{attribute addProperty BoxType "EK1100-0000-0018"}
{attribute addProperty Id "Beckhoff_EL34xxEK1122Beckhoff_EL34xxEK1122_54E02F3C162A_0001_EL3403_0000_0017EL3403_CEBF0ECD61677A_0002_EL3403_0000_0018EL3403_0856E9FD61677A_0003_EL3403_0000_0019EL3403_0856E9FD61677A_0004_EL3403_0000_0020EL3403_0856E9FD61677A_0005_EL3403_0000_0021EL3403_0856E9FD61677A_0006_EL3403_0000_0022EL3403_26274D9958473A_0007_EL3403_0000_0023EL3403_26274D9958473A_0008_EL3403_0010_0017EL3403_CEBF0ECD61677A_0009_EL3403_0010_0018EL3403_0856E9FD61677A_0010_EL3403_0010_0019EL3403_0856E9FD61677A_0011_EL3403_0010_0020EL3403_0856E9FD61677A_0012_EL3403_0010_0021EL3403_0856E9FD61677A_0013_EL3403_0010_0022EL3403_26274D9958473A_0014_EL3403_0010_0023EL3403_26274D9958473A_0015_EL3403_0010_0024EL3403_26274D9958473A_0016_EL3403_0026_0017EL3403_CEBF0ECD61677A_0017_EL3403_0026_0018EL3403_0856E9FD61677A_0018_EL3403_0026_0019EL3403_0856E9FD61677A_0019_EL3403_0026_0020EL3403_0856E9FD61677A_0020_EL3403_0026_0021EL3403_0856E9FD61677A_0021_EL3403_0026_0022EL3403_26274D9958473A_0022_EL3403_0026_0023EL3403_26274D9958473A_0023_EL3403_0026_0024EL3403_26274D9958473A_0024_EL3403_0100_0017EL3403_CEBF0ECD61677A_0025_EL3403_0100_0018EL3403_0856E9FD61677A_0026_EL3403_0100_0019EL3403_0856E9FD61677A_0027_EL3403_0100_0020EL3403_0856E9FD61677A_0028_EL3403_0100_0021EL3403_0856E9FD61677A_0029_EL3403_0100_0022EL3403_26274D9958473A_0030_EL3403_0100_0023EL3403_26274D9958473A_0031_EL3403_0100_0024EL3403_26274D9958473A_0032_EL3403_0111_0017EL3403_CEBF0ECD61677A_0033_EL3403_0111_0018EL3403_0856E9FD61677A_0034_EL3403_0111_0019EL3403_0856E9FD61677A_0035_EL3403_0111_0020EL3403_0856E9FD61677A_0036_EL3403_0111_0021EL3403_0856E9FD61677A_0037_EL3403_0111_0022EL3403_26274D9958473A_0038_EL3403_0111_0023EL3403_26274D9958473A_0039_EL3403_0111_0024EL3403_26274D9958473A_0040_EL3403_0126_0017EL3403_CEBF0ECD61677A_0041_EL3403_0126_0018EL3403_0856E9FD61677A_0042_EL3403_0126_0019EL3403_0856E9FD61677A_0043_EL3403_0126_0020EL3403_0856E9FD61677A_0044_EL3403_0126_0021EL3403_0856E9FD61677A_0045_EL3403_0126_0022EL3403_26274D9958473A_0046_EL3403_0126_0023EL3403_26274D9958473A_0047_EL3403_0126_0024EL3403_26274D9958473A_0048_EL3403_0333_0023EL3403_26274D9958473A_0049_EL3403_0333_0024EL3403_26274D9958473A_0050_EL3413_0000_0016EL3413_446C23E765682A_0051_EL3413_0000_0017EL3413_446C23E765682A_0052_EL3413_0000_0018EL3413_446C23E765682A_0053_EL3413_0000_0019EL3413_7AF41FD265682A_0054_EL3413_0000_0020EL3413_7AF41FD265682A_0055_EL3413_0001_0016EL3413_7AF41FD265682A_0056_EL3413_0001_0017EL3413_7AF41FD265682A_0057_EL3413_0120_0017EL3413_446C23E765682A_0058_EL3413_0001_0018EL3413_7AF41FD265682A_0059_EL3413_0120_0018EL3413_7AF41FD265682A_0060_EL3413_0120_0019EL3413_7AF41FD265682A_0061_EL3423_0000_0016EL3423_A72AC4D21520190A_0062_EL3423_0000_0017EL3423_51F4B0921520190A_0063_EL3423_0000_0018EL3423_51F4B0921520190A_0064_EL3423_0000_0019EL3423_51F4B0921520190A_0065_EL3423_0000_0020EL3423_5F1A409A944118A_0066_EL3423_0000_0021EL3423_5F1A409A944118A_0067_EL3433_0000_0016EL3433_7AF41FD265682A_0068_EL3433_0000_0017EL3433_7AF41FD265682A_0069_EL3433_0000_0018EL3433_7AF41FD265682A_0070_EL3443_0000_0016EL3443_FBA7AEAF1664208A_0071_EL3443_0000_0017EL3443_A40FED4E1664208A_0072_EL3443_0000_0018EL3443_A40FED4E1664208A_0073_EL3443_0000_0019EL3443_A40FED4E1664208A_0074_EL3443_0000_0020EL3443_FBA7AEAF1664208A_0075_EL3443_0000_0021EL3443_FBA7AEAF1664208A_0076_EL3443_0010_0016EL3443_FBA7AEAF1664208A_0077_EL3443_0010_0017EL3443_A40FED4E1664208A_0078_EL3443_0010_0018EL3443_A40FED4E1664208A_0079_EL3443_0010_0019EL3443_A40FED4E1664208A_0080_EL3443_0010_0020EL3443_FBA7AEAF1664208A_0081_EL3443_0010_0021EL3443_FBA7AEAF1664208A_0082_EL3443_0011_0018EL3443_A40FED4E1664208A_0083_EL3443_0011_0019EL3443_A40FED4E1664208A_0084_EL3443_0011_0020EL3443_FBA7AEAF1664208A_0085_EL3443_0011_0021EL3443_FBA7AEAF1664208A_0086_EL3443_0013_0018EL3443_A40FED4E1664208A_0087_EL3443_0013_0019EL3443_A40FED4E1664208A_0088_EL3443_0013_0020EL3443_FBA7AEAF1664208A_0089_EL3443_0013_0021EL3443_FBA7AEAF1664208A_0090_EL3446_0000_0016EL3446_CF28416359274A_0091_EL3446_0000_0017EL3446_CF28416359274A_0092_EL3453_0000_0017EL3453_04D436851216152A_0093_EL3453_0000_0018EL3453_0BDF0D211208151A_0094_EL3453_0000_0019EL3453_0BDF0D211208151A_0095_EL3453_0000_0020EL3453_04D436851216152A_0096_EL3453_0000_0021EL3453_04D436851216152A_0097_EL3453_0100_0021EL3453_04D436851216152A_0098_EL3483_0000_0016EL3483_4775AA5232841A_0099_EL3483_0000_0017EL3483_4775AA5232841A_0100_EL3483_0000_0018EL3483_4775AA5232841A_0101_EL3483_0000_0019EL3483_4775AA5232841A_0102_EL3483_0000_0020EL3483_4775AA5232841A_0103_EL3483_0000_0021EL3483_4775AA5232841A_0104_EL3483_0060_0018EL3483_52D9841A52065A_0105_EL3483_0060_0019EL3483_52D9841A52065A_0106_EL3483_0060_0020EL3483_FF2A77B352065A_0107_EL3483_0060_0021EL3483_FF2A77B352065"}
{attribute addProperty CRC "1912410272"}
{attribute addProperty SizeInBites "92536"}
{attribute addProperty SizeInBytes "11567"}
TYPE Beckhoff_EL34xx_71FD10A0 EXTENDS EK1100_179A0949 :
STRUCT
	{attribute addProperty Name "Beckhoff_EL34xxEK1122"}
	Beckhoff_EL34xxEK1122 : Beckhoff_EL34xxEK1122_54E02F3C;
	{attribute addProperty Name "A_0001_EL3403_0000_0017"}
	A_0001_EL3403_0000_0017 : EL3403_CEBF0ECD;
	{attribute addProperty Name "A_0002_EL3403_0000_0018"}
	A_0002_EL3403_0000_0018 : EL3403_0856E9FD;
	{attribute addProperty Name "A_0003_EL3403_0000_0019"}
	A_0003_EL3403_0000_0019 : EL3403_0856E9FD;
	{attribute addProperty Name "A_0004_EL3403_0000_0020"}
	A_0004_EL3403_0000_0020 : EL3403_0856E9FD;
	{attribute addProperty Name "A_0005_EL3403_0000_0021"}
	A_0005_EL3403_0000_0021 : EL3403_0856E9FD;
	{attribute addProperty Name "A_0006_EL3403_0000_0022"}
	A_0006_EL3403_0000_0022 : EL3403_26274D99;
	{attribute addProperty Name "A_0007_EL3403_0000_0023"}
	A_0007_EL3403_0000_0023 : EL3403_26274D99;
	{attribute addProperty Name "A_0008_EL3403_0010_0017"}
	A_0008_EL3403_0010_0017 : EL3403_CEBF0ECD;
	{attribute addProperty Name "A_0009_EL3403_0010_0018"}
	A_0009_EL3403_0010_0018 : EL3403_0856E9FD;
	{attribute addProperty Name "A_0010_EL3403_0010_0019"}
	A_0010_EL3403_0010_0019 : EL3403_0856E9FD;
	{attribute addProperty Name "A_0011_EL3403_0010_0020"}
	A_0011_EL3403_0010_0020 : EL3403_0856E9FD;
	{attribute addProperty Name "A_0012_EL3403_0010_0021"}
	A_0012_EL3403_0010_0021 : EL3403_0856E9FD;
	{attribute addProperty Name "A_0013_EL3403_0010_0022"}
	A_0013_EL3403_0010_0022 : EL3403_26274D99;
	{attribute addProperty Name "A_0014_EL3403_0010_0023"}
	A_0014_EL3403_0010_0023 : EL3403_26274D99;
	{attribute addProperty Name "A_0015_EL3403_0010_0024"}
	A_0015_EL3403_0010_0024 : EL3403_26274D99;
	{attribute addProperty Name "A_0016_EL3403_0026_0017"}
	A_0016_EL3403_0026_0017 : EL3403_CEBF0ECD;
	{attribute addProperty Name "A_0017_EL3403_0026_0018"}
	A_0017_EL3403_0026_0018 : EL3403_0856E9FD;
	{attribute addProperty Name "A_0018_EL3403_0026_0019"}
	A_0018_EL3403_0026_0019 : EL3403_0856E9FD;
	{attribute addProperty Name "A_0019_EL3403_0026_0020"}
	A_0019_EL3403_0026_0020 : EL3403_0856E9FD;
	{attribute addProperty Name "A_0020_EL3403_0026_0021"}
	A_0020_EL3403_0026_0021 : EL3403_0856E9FD;
	{attribute addProperty Name "A_0021_EL3403_0026_0022"}
	A_0021_EL3403_0026_0022 : EL3403_26274D99;
	{attribute addProperty Name "A_0022_EL3403_0026_0023"}
	A_0022_EL3403_0026_0023 : EL3403_26274D99;
	{attribute addProperty Name "A_0023_EL3403_0026_0024"}
	A_0023_EL3403_0026_0024 : EL3403_26274D99;
	{attribute addProperty Name "A_0024_EL3403_0100_0017"}
	A_0024_EL3403_0100_0017 : EL3403_CEBF0ECD;
	{attribute addProperty Name "A_0025_EL3403_0100_0018"}
	A_0025_EL3403_0100_0018 : EL3403_0856E9FD;
	{attribute addProperty Name "A_0026_EL3403_0100_0019"}
	A_0026_EL3403_0100_0019 : EL3403_0856E9FD;
	{attribute addProperty Name "A_0027_EL3403_0100_0020"}
	A_0027_EL3403_0100_0020 : EL3403_0856E9FD;
	{attribute addProperty Name "A_0028_EL3403_0100_0021"}
	A_0028_EL3403_0100_0021 : EL3403_0856E9FD;
	{attribute addProperty Name "A_0029_EL3403_0100_0022"}
	A_0029_EL3403_0100_0022 : EL3403_26274D99;
	{attribute addProperty Name "A_0030_EL3403_0100_0023"}
	A_0030_EL3403_0100_0023 : EL3403_26274D99;
	{attribute addProperty Name "A_0031_EL3403_0100_0024"}
	A_0031_EL3403_0100_0024 : EL3403_26274D99;
	{attribute addProperty Name "A_0032_EL3403_0111_0017"}
	A_0032_EL3403_0111_0017 : EL3403_CEBF0ECD;
	{attribute addProperty Name "A_0033_EL3403_0111_0018"}
	A_0033_EL3403_0111_0018 : EL3403_0856E9FD;
	{attribute addProperty Name "A_0034_EL3403_0111_0019"}
	A_0034_EL3403_0111_0019 : EL3403_0856E9FD;
	{attribute addProperty Name "A_0035_EL3403_0111_0020"}
	A_0035_EL3403_0111_0020 : EL3403_0856E9FD;
	{attribute addProperty Name "A_0036_EL3403_0111_0021"}
	A_0036_EL3403_0111_0021 : EL3403_0856E9FD;
	{attribute addProperty Name "A_0037_EL3403_0111_0022"}
	A_0037_EL3403_0111_0022 : EL3403_26274D99;
	{attribute addProperty Name "A_0038_EL3403_0111_0023"}
	A_0038_EL3403_0111_0023 : EL3403_26274D99;
	{attribute addProperty Name "A_0039_EL3403_0111_0024"}
	A_0039_EL3403_0111_0024 : EL3403_26274D99;
	{attribute addProperty Name "A_0040_EL3403_0126_0017"}
	A_0040_EL3403_0126_0017 : EL3403_CEBF0ECD;
	{attribute addProperty Name "A_0041_EL3403_0126_0018"}
	A_0041_EL3403_0126_0018 : EL3403_0856E9FD;
	{attribute addProperty Name "A_0042_EL3403_0126_0019"}
	A_0042_EL3403_0126_0019 : EL3403_0856E9FD;
	{attribute addProperty Name "A_0043_EL3403_0126_0020"}
	A_0043_EL3403_0126_0020 : EL3403_0856E9FD;
	{attribute addProperty Name "A_0044_EL3403_0126_0021"}
	A_0044_EL3403_0126_0021 : EL3403_0856E9FD;
	{attribute addProperty Name "A_0045_EL3403_0126_0022"}
	A_0045_EL3403_0126_0022 : EL3403_26274D99;
	{attribute addProperty Name "A_0046_EL3403_0126_0023"}
	A_0046_EL3403_0126_0023 : EL3403_26274D99;
	{attribute addProperty Name "A_0047_EL3403_0126_0024"}
	A_0047_EL3403_0126_0024 : EL3403_26274D99;
	{attribute addProperty Name "A_0048_EL3403_0333_0023"}
	A_0048_EL3403_0333_0023 : EL3403_26274D99;
	{attribute addProperty Name "A_0049_EL3403_0333_0024"}
	A_0049_EL3403_0333_0024 : EL3403_26274D99;
	{attribute addProperty Name "A_0050_EL3413_0000_0016"}
	A_0050_EL3413_0000_0016 : EL3413_446C23E7;
	{attribute addProperty Name "A_0051_EL3413_0000_0017"}
	A_0051_EL3413_0000_0017 : EL3413_446C23E7;
	{attribute addProperty Name "A_0052_EL3413_0000_0018"}
	A_0052_EL3413_0000_0018 : EL3413_446C23E7;
	{attribute addProperty Name "A_0053_EL3413_0000_0019"}
	A_0053_EL3413_0000_0019 : EL3413_7AF41FD2;
	{attribute addProperty Name "A_0054_EL3413_0000_0020"}
	A_0054_EL3413_0000_0020 : EL3413_7AF41FD2;
	{attribute addProperty Name "A_0055_EL3413_0001_0016"}
	A_0055_EL3413_0001_0016 : EL3413_7AF41FD2;
	{attribute addProperty Name "A_0056_EL3413_0001_0017"}
	A_0056_EL3413_0001_0017 : EL3413_7AF41FD2;
	{attribute addProperty Name "A_0057_EL3413_0120_0017"}
	A_0057_EL3413_0120_0017 : EL3413_446C23E7;
	{attribute addProperty Name "A_0058_EL3413_0001_0018"}
	A_0058_EL3413_0001_0018 : EL3413_7AF41FD2;
	{attribute addProperty Name "A_0059_EL3413_0120_0018"}
	A_0059_EL3413_0120_0018 : EL3413_7AF41FD2;
	{attribute addProperty Name "A_0060_EL3413_0120_0019"}
	A_0060_EL3413_0120_0019 : EL3413_7AF41FD2;
	{attribute addProperty Name "A_0061_EL3423_0000_0016"}
	A_0061_EL3423_0000_0016 : EL3423_A72AC4D2;
	{attribute addProperty Name "A_0062_EL3423_0000_0017"}
	A_0062_EL3423_0000_0017 : EL3423_51F4B092;
	{attribute addProperty Name "A_0063_EL3423_0000_0018"}
	A_0063_EL3423_0000_0018 : EL3423_51F4B092;
	{attribute addProperty Name "A_0064_EL3423_0000_0019"}
	A_0064_EL3423_0000_0019 : EL3423_51F4B092;
	{attribute addProperty Name "A_0065_EL3423_0000_0020"}
	A_0065_EL3423_0000_0020 : EL3423_5F1A409A;
	{attribute addProperty Name "A_0066_EL3423_0000_0021"}
	A_0066_EL3423_0000_0021 : EL3423_5F1A409A;
	{attribute addProperty Name "A_0067_EL3433_0000_0016"}
	A_0067_EL3433_0000_0016 : EL3433_7AF41FD2;
	{attribute addProperty Name "A_0068_EL3433_0000_0017"}
	A_0068_EL3433_0000_0017 : EL3433_7AF41FD2;
	{attribute addProperty Name "A_0069_EL3433_0000_0018"}
	A_0069_EL3433_0000_0018 : EL3433_7AF41FD2;
	{attribute addProperty Name "A_0070_EL3443_0000_0016"}
	A_0070_EL3443_0000_0016 : EL3443_FBA7AEAF;
	{attribute addProperty Name "A_0071_EL3443_0000_0017"}
	A_0071_EL3443_0000_0017 : EL3443_A40FED4E;
	{attribute addProperty Name "A_0072_EL3443_0000_0018"}
	A_0072_EL3443_0000_0018 : EL3443_A40FED4E;
	{attribute addProperty Name "A_0073_EL3443_0000_0019"}
	A_0073_EL3443_0000_0019 : EL3443_A40FED4E;
	{attribute addProperty Name "A_0074_EL3443_0000_0020"}
	A_0074_EL3443_0000_0020 : EL3443_FBA7AEAF;
	{attribute addProperty Name "A_0075_EL3443_0000_0021"}
	A_0075_EL3443_0000_0021 : EL3443_FBA7AEAF;
	{attribute addProperty Name "A_0076_EL3443_0010_0016"}
	A_0076_EL3443_0010_0016 : EL3443_FBA7AEAF;
	{attribute addProperty Name "A_0077_EL3443_0010_0017"}
	A_0077_EL3443_0010_0017 : EL3443_A40FED4E;
	{attribute addProperty Name "A_0078_EL3443_0010_0018"}
	A_0078_EL3443_0010_0018 : EL3443_A40FED4E;
	{attribute addProperty Name "A_0079_EL3443_0010_0019"}
	A_0079_EL3443_0010_0019 : EL3443_A40FED4E;
	{attribute addProperty Name "A_0080_EL3443_0010_0020"}
	A_0080_EL3443_0010_0020 : EL3443_FBA7AEAF;
	{attribute addProperty Name "A_0081_EL3443_0010_0021"}
	A_0081_EL3443_0010_0021 : EL3443_FBA7AEAF;
	{attribute addProperty Name "A_0082_EL3443_0011_0018"}
	A_0082_EL3443_0011_0018 : EL3443_A40FED4E;
	{attribute addProperty Name "A_0083_EL3443_0011_0019"}
	A_0083_EL3443_0011_0019 : EL3443_A40FED4E;
	{attribute addProperty Name "A_0084_EL3443_0011_0020"}
	A_0084_EL3443_0011_0020 : EL3443_FBA7AEAF;
	{attribute addProperty Name "A_0085_EL3443_0011_0021"}
	A_0085_EL3443_0011_0021 : EL3443_FBA7AEAF;
	{attribute addProperty Name "A_0086_EL3443_0013_0018"}
	A_0086_EL3443_0013_0018 : EL3443_A40FED4E;
	{attribute addProperty Name "A_0087_EL3443_0013_0019"}
	A_0087_EL3443_0013_0019 : EL3443_A40FED4E;
	{attribute addProperty Name "A_0088_EL3443_0013_0020"}
	A_0088_EL3443_0013_0020 : EL3443_FBA7AEAF;
	{attribute addProperty Name "A_0089_EL3443_0013_0021"}
	A_0089_EL3443_0013_0021 : EL3443_FBA7AEAF;
	{attribute addProperty Name "A_0090_EL3446_0000_0016"}
	A_0090_EL3446_0000_0016 : EL3446_CF284163;
	{attribute addProperty Name "A_0091_EL3446_0000_0017"}
	A_0091_EL3446_0000_0017 : EL3446_CF284163;
	{attribute addProperty Name "A_0092_EL3453_0000_0017"}
	A_0092_EL3453_0000_0017 : EL3453_04D43685;
	{attribute addProperty Name "A_0093_EL3453_0000_0018"}
	A_0093_EL3453_0000_0018 : EL3453_0BDF0D21;
	{attribute addProperty Name "A_0094_EL3453_0000_0019"}
	A_0094_EL3453_0000_0019 : EL3453_0BDF0D21;
	{attribute addProperty Name "A_0095_EL3453_0000_0020"}
	A_0095_EL3453_0000_0020 : EL3453_04D43685;
	{attribute addProperty Name "A_0096_EL3453_0000_0021"}
	A_0096_EL3453_0000_0021 : EL3453_04D43685;
	{attribute addProperty Name "A_0097_EL3453_0100_0021"}
	A_0097_EL3453_0100_0021 : EL3453_04D43685;
	{attribute addProperty Name "A_0098_EL3483_0000_0016"}
	A_0098_EL3483_0000_0016 : EL3483_4775AA52;
	{attribute addProperty Name "A_0099_EL3483_0000_0017"}
	A_0099_EL3483_0000_0017 : EL3483_4775AA52;
	{attribute addProperty Name "A_0100_EL3483_0000_0018"}
	A_0100_EL3483_0000_0018 : EL3483_4775AA52;
	{attribute addProperty Name "A_0101_EL3483_0000_0019"}
	A_0101_EL3483_0000_0019 : EL3483_4775AA52;
	{attribute addProperty Name "A_0102_EL3483_0000_0020"}
	A_0102_EL3483_0000_0020 : EL3483_4775AA52;
	{attribute addProperty Name "A_0103_EL3483_0000_0021"}
	A_0103_EL3483_0000_0021 : EL3483_4775AA52;
	{attribute addProperty Name "A_0104_EL3483_0060_0018"}
	A_0104_EL3483_0060_0018 : EL3483_52D9841A;
	{attribute addProperty Name "A_0105_EL3483_0060_0019"}
	A_0105_EL3483_0060_0019 : EL3483_52D9841A;
	{attribute addProperty Name "A_0106_EL3483_0060_0020"}
	A_0106_EL3483_0060_0020 : EL3483_FF2A77B3;
	{attribute addProperty Name "A_0107_EL3483_0060_0021"}
	A_0107_EL3483_0060_0021 : EL3483_FF2A77B3;
END_STRUCT
END_TYPE

(* stored: Version 1.2.0.0, ProductVersion 3.1.4024.9
   DUT Beckhoff_EL34xx_71FD10A0: Id {4eb58c06-66ee-4181-971f-a273191d532b} *)
